FUNCTION_BLOCK TcoSegmentDoor_Close EXTENDS TcoCore.TcoSequencer
VAR
	_o : TcoCore.TcoSequencerObserver(THIS^);	
	_dialog : TcoCore.TcoDialog(THIS^);
END_VAR

{error 'Eigenschaftenimplementierung hinzufügen oder Eigenschaft löschen, um die Basisimplementierung zu verwenden'}
PROPERTY Context : TcoCore.ITcoContext
GET
END_GET
END_PROPERTY

{error 'Eigenschaftenimplementierung hinzufügen oder Eigenschaft löschen, um die Basisimplementierung zu verwenden'}
(*~
	<docu>
		<summary>
			Gets the information about the current step.						
		</summary>				
	</docu>	
~*)
PROPERTY CurrentStep : REFERENCE TO TcoCore.StepDetails
GET
END_GET
END_PROPERTY

{error 'Eigenschaftenimplementierung hinzufügen oder Eigenschaft löschen, um die Basisimplementierung zu verwenden'}
PROPERTY Identity : ULINT
GET
END_GET
END_PROPERTY

{error 'Eigenschaftenimplementierung hinzufügen oder Eigenschaft löschen, um die Basisimplementierung zu verwenden'}
PROPERTY IsAutoRestoreEnabled : BOOL
GET
END_GET
END_PROPERTY

{error 'Eigenschaftenimplementierung hinzufügen oder Eigenschaft löschen, um die Basisimplementierung zu verwenden'}
PROPERTY IsFreshState : BOOL
GET
END_GET
END_PROPERTY

{error 'Eigenschaftenimplementierung hinzufügen oder Eigenschaft löschen, um die Basisimplementierung zu verwenden'}
PROPERTY LastStateChangeCycle : ULINT
GET
END_GET
END_PROPERTY

{warning 'Methodenimplementierung hinzufügen'}
(*~
	<docu>
		<summary>
			Main method of the sequener. Custom code needs to be placed here. The sequencer is executed by call of **Instance.Run()** method.
			This method is abstract, and it must be overridden in derived block.
		</summary>
	</docu>
~*)
METHOD PROTECTED Main : BOOL
END_METHOD

{error 'Eigenschaftenimplementierung hinzufügen oder Eigenschaft löschen, um die Basisimplementierung zu verwenden'}
PROPERTY ModeController : TcoCore.ITcoSequencerModeController
GET
END_GET
END_PROPERTY

{warning 'Methodenimplementierung hinzufügen'}
METHOD MoveNext : BOOL
END_METHOD

{warning 'Methodenimplementierung hinzufügen'}
METHOD Restore : TcoCore.ITcoRestorable
END_METHOD

{warning 'Methodenimplementierung hinzufügen'}
METHOD RestoreObject : TcoCore.ITcoObjectRestorer
VAR_INPUT
	Obj	: TcoCore.ITcoRestorable;
END_VAR
END_METHOD

{warning 'Methodenimplementierung hinzufügen'}
METHOD Retry : BOOL
VAR_INPUT
	inFromState	: INT;
END_VAR
END_METHOD

{error 'Eigenschaftenimplementierung hinzufügen oder Eigenschaft löschen, um die Basisimplementierung zu verwenden'}
PROPERTY State : INT
GET
END_GET
END_PROPERTY

{warning 'Methodenimplementierung hinzufügen'}
METHOD Terminate : BOOL
END_METHOD

END_FUNCTION_BLOCK

(* stored: Version 1.1.0.1
   POU TcoSegmentDoor_Close: Id {4f1e7c88-97a5-4883-b1d3-e7f7f73a8c0b}, SpecialFunc None
   Property Context: Id {036130e7-03f6-4401-b264-b8f4f275ce33}
   Get Get: Id {ca87d0d3-e205-4e93-b725-844dac76e36a}
   Property CurrentStep: Id {3c1762ca-4f0d-4b77-b81f-d95962b69969}
   Get Get: Id {06e767db-d1be-4894-8a3e-34d6a4e30c17}
   Property Identity: Id {6c688134-13b1-4f94-b023-7153aaf3ad67}
   Get Get: Id {d76293e8-3be7-4128-992f-9a6f5771ca8b}
   Property IsAutoRestoreEnabled: Id {4179be0b-8f38-4e5d-bdd0-c9cd9111d948}
   Get Get: Id {b1a17375-9ded-43e7-a35c-747bb9e3c6c5}
   Property IsFreshState: Id {1a8fc16c-7241-42fd-bd49-1b3ef733029a}
   Get Get: Id {3bb57f92-d416-4ed9-86c6-41148f2d4b53}
   Property LastStateChangeCycle: Id {0f2d927a-59ca-46d8-9793-eef8b0211f0e}
   Get Get: Id {8c37f72a-d4e6-48d1-8ae9-b55fa5cd1cf6}
   Method Main: Id {89467f8d-8a59-4d01-b068-bcd5624f7577}
   Property ModeController: Id {a657e86b-ac68-4b0f-add5-c0373791c437}
   Get Get: Id {af1b9034-9afb-43c7-978f-cc59cf099bc3}
   Method MoveNext: Id {90c5dbb8-eb0e-40aa-a8d2-f8e505067a60}
   Method Restore: Id {3bc01d8c-9856-46c8-8a37-c9739d852b77}
   Method RestoreObject: Id {c68e033a-d176-4d2a-a3f9-486778096ccb}
   Method Retry: Id {e7b9d5cf-949e-480e-83a3-425f09aa96f6}
   Property State: Id {39d97dc5-ee8b-4204-86f8-6e5423ba3960}
   Get Get: Id {89f7fbcd-9547-4c9d-9deb-64c20e236161}
   Method Terminate: Id {9c858178-d788-4632-81d6-6074a2018404} *)
